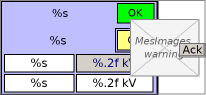
VISUALIZATION VISU_HT_GENIUS_ETH  // 206x95
VAR_IN_OUT
	m_Input_SOURCE : BLOCK_SOURCE_GENIUS_ETHERCAT;
END_VAR
    Rectangle (0,0 158x95)
    Rectangle (3,30 110x21), "%s", text list: 'TextList_Evap', text index: 3
    Rectangle (117,3 37x20), "NOK", invisible if: NOT m_Input_SOURCE.STATE_NOK
    Rectangle (117,30 37x20), "OFF", invisible if: m_Input_SOURCE.STATE_HV OR m_Input_SOURCE.STATE_HV_ON
    Rectangle (117,3 37x20), "OK", invisible if: m_Input_SOURCE.STATE_NOK
    Rectangle (117,30 37x20), "ON", invisible if: NOT m_Input_SOURCE.STATE_HV AND NOT m_Input_SOURCE.STATE_HV_ON
    RoundedRectangle (4,54 70x18), "%s", invisible if: Global_Variables.MACHINE.State_manu, text list: 'TextList_Evap', text index: 4
    RoundedRectangle (76,54 77x18), "%.2f kV", text variable: m_Input_SOURCE.STATE_TENSION, invisible if: Global_Variables.MACHINE.State_manu
    Rectangle (117,30 37x20), "ON", invisible if: m_Input_SOURCE.STATE_HV_ON OR NOT m_Input_SOURCE.STATE_HV
    Rectangle (0,3 120x21), "%s", text variable: m_Input_SOURCE.MNEMO
    Polyline (7,35)
    RoundedRectangle (4,74 70x18), "%s", invisible if: NOT Global_Variables.PRG_USER.ACTU_USER.MAINTENANCE OR NOT MACHINE.State_manu, text list: 'TextList_Evap', text index: 4
    RoundedRectangle (76,74 77x18), "%.2f kV", text variable: m_Input_SOURCE.PRM_TENSION, invisible if: NOT Global_Variables.PRG_USER.ACTU_USER.MAINTENANCE OR NOT MACHINE.STATE_Manu
        OnMouseDown: write the text variable via VisuDialogs.Numpad, min 7, max 10
    Rectangle (115,28 41x24), invisible if: NOT m_Input_SOURCE.HV.AUTOR_ON_IHM AND NOT m_Input_SOURCE.HV.AUTOR_OFF_IHM, input disabled if: (NOT m_Input_SOURCE.HV.AUTOR_ON_IHM AND NOT m_Input_SOURCE.HV.AUTOR_OFF_IHM) OR NOT PRG_User.ACTU_USER.MAINTENANCE
        tap m_Input_SOURCE.HV.M_On
    Image (130,19 69x57), invisible if: NOT m_Input_SOURCE.HV.STATE_Nok AND NOT m_Input_SOURCE.DEF_Source.DEF AND NOT m_Input_SOURCE.DEF_Communication.DEF AND NOT m_Input_SOURCE.DEF_HV.DEF, image: MesImages.warning
    Button (179,43 27x14), "Ack", invisible if: NOT m_Input_SOURCE.HV.STATE_Nok AND NOT m_Input_SOURCE.DEF_Source.DEF AND NOT m_Input_SOURCE.DEF_Communication.DEF AND NOT m_Input_SOURCE.DEF_HV.DEF
        tap m_Input_SOURCE.M_Ack
END_VISUALIZATION

(* stored: Version 1.1.0.1, ProductVersion 3.1.4024.10
   Visu VISU_HT_GENIUS_ETH: Id {f700acc2-8dea-4f10-bb0d-3867608cd5a1} *)
